INTERFACE I_UniversalMotor

METHOD Abort : BOOL
VAR_INPUT
END_VAR
END_METHOD

PROPERTY ActualPosition : LREAL
GET
END_GET
END_PROPERTY

PROPERTY AxisReference : AXIS_REF
GET
END_GET
END_PROPERTY

METHOD Couple : BOOL
VAR_INPUT

END_VAR

VAR

END_VAR
END_METHOD

PROPERTY Coupleable : BOOL
GET
END_GET
SET
END_SET
END_PROPERTY

PROPERTY Coupled : BOOL
GET
END_GET
END_PROPERTY

METHOD Decouple : BOOL
VAR_INPUT
END_VAR
VAR
END_VAR
END_METHOD

METHOD Home : BOOL // Start axis homing
VAR_INPUT
END_VAR
END_METHOD

PROPERTY Homed : BOOL
GET
END_GET
END_PROPERTY

PROPERTY Homingable : BOOL
GET
END_GET
SET
END_SET
END_PROPERTY

METHOD Init : BOOL
VAR_INPUT
END_VAR
END_METHOD

PROPERTY Initialized : BOOL
GET
END_GET
END_PROPERTY

METHOD Jog : BOOL
VAR_INPUT
	Distance	:	LREAL;
END_VAR
END_METHOD

PROPERTY MotorName : STRING
GET
END_GET
SET
END_SET
END_PROPERTY

METHOD MoveAbsolute : BOOL // Do action 2 request, for instance: 'Pick and place unit' change tool (additional inputs needed)
VAR_INPUT
	Position : LREAL;
END_VAR
END_METHOD

METHOD Reset : BOOL
VAR_INPUT
END_VAR
END_METHOD

PROPERTY Unit : STRING
GET
END_GET
SET
END_SET
END_PROPERTY

END_INTERFACE

(* stored: Version 1.1.0.1, ProductVersion 3.1.4024.12
   Itf I_UniversalMotor: Id {95ea5372-be3d-45e1-9d49-97657d69cbe0}
   Method Abort: Id {41ef6a92-9d3e-44b0-ac70-e72ab78cbf8c}
   Property ActualPosition: Id {bdcc4591-5f17-41e2-afcb-d062baca1b15}
   Get Get: Id {042ae297-1ed6-41ce-b1c7-60b45c5a1b9c}
   Property AxisReference: Id {9f5d9b85-41e4-4674-89f4-8c092f3d48ec}
   Get Get: Id {ca5aaa11-ee4b-45d1-8d24-e6b2262f8cbc}
   Method Couple: Id {33ff9662-8bdf-4838-a0fb-391f702fd051}
   Property Coupleable: Id {f4a27231-e466-4cc2-be4e-b981a7c7d6a6}
   Get Get: Id {931fa3ba-8bac-4ba3-9ac7-61833283be2f}
   Set Set: Id {ac28e13a-d0a4-4ebd-9b00-71b6aa5ebcbd}
   Property Coupled: Id {d7cc03fc-5a61-48d0-904a-967828847224}
   Get Get: Id {c5089489-827c-4844-b0ef-a5cdc4868251}
   Method Decouple: Id {6df1250b-4080-44e8-ab6b-63e423e87208}
   Method Home: Id {a958eb08-04f8-4467-ad60-342dbeb4cb8a}
   Property Homed: Id {3f29323e-79f2-445c-b593-2ecda2f6bf32}
   Get Get: Id {1cae9f13-6b6a-4fed-9cb9-8e7ff2b308c3}
   Property Homingable: Id {31bdf3d2-4dcc-4dfd-929d-caab6e58e871}
   Get Get: Id {b52effb0-cc7e-4a53-9d17-5050e2b3e5b5}
   Set Set: Id {4f92f0f5-a196-4d0b-89e6-49c7109e2d12}
   Method Init: Id {0b8cd39f-02f7-476d-9199-5d7119c1c212}
   Property Initialized: Id {eb994419-eac6-4b52-8ef4-41f3857e16cf}
   Get Get: Id {5e49cecf-31fb-4190-9689-3950da99505c}
   Method Jog: Id {95b8d47c-45bc-4fc1-80ea-5784b7382dc0}
   Property MotorName: Id {2e4bf95e-5be0-4191-9fe4-869e161b9c62}
   Get Get: Id {c1e2e84f-3a2a-4510-a06a-d7cc60afdbb0}
   Set Set: Id {1fb93800-79e6-48cb-8f9b-a5b47db29813}
   Method MoveAbsolute: Id {e089bf2c-4a92-4acb-8a76-61430383c3f3}
   Method Reset: Id {68abb08b-f886-4a29-8cc3-a9583cd195a7}
   Property Unit: Id {06983b9e-8e66-4409-9f5a-827371225648}
   Get Get: Id {d7b49bac-d72a-4073-8273-d38c230dcc33}
   Set Set: Id {740f0242-9622-4ced-8c6b-95645d2cfb9f} *)
